{attribute 'qualified_only'}
{attribute 'strict'}
{attribute 'to_string'}
TYPE LinearAxis_e :
(
    ST110_01Y,
    ST110_02Z,
    ST110_03Z,
    ST110_04Z,
    ST115_01Y,
    ST115_02Z,
    ST115_03Z,
    ST115_04Z,
    ST120_01Y,
    ST120_02Z,
    _max
);
END_TYPE

(* stored: Version 1.1.0.1, ProductVersion 3.1.4024.6
   DUT LinearAxis_e: Id {969b3950-fd06-4754-aef9-7edb95613f8d} *)
